PROGRAM LedControl
VAR
	
	
	
	
END_VAR

END_PROGRAM

(* stored: Version 1.1.0.1, ProductVersion 3.1.4024.14
   POU LedControl: Id {090f8d70-b946-43d6-a2ea-e3b753c1d298}, SpecialFunc None *)
